// TIA Portal V20 export
FUNCTION_BLOCK "FB_LaserMeasureZoneSwitch"   // FB417, SCL
{ S7_Optimized_Access := 'TRUE' }
// stored: AutoNumber false, MemoryReserve 100, SetENOAutomatically false
   VAR RETAIN
      sMeasure1 : Bool;   // Limit sw Measure 1 / Axes are on Area Measure station 1
      sMeasure2 : Bool;   // Limit sw Measure 2 / Axes are on Area Measure station 2
      sLaser1 : Bool;   // Condition Laser 1 / Gate for going to area laser Station 1
      sLaser2 : Bool;   // Condition Laser 2 / Gate for going to area laser Station 2
      sLaserArea1Req : Bool;   // Laser area 1 request / Ask for going to laser Area Station 1
      sLaserArea2Req : Bool;   // Laser area 2 request / Ask for going to laser Area Station 2
      sCuttingArea1Req : Bool;   // Cutting 1 request / Axe X1 enter to laser Area
      sCuttingArea2Req : Bool;   // Cutting 2 request / Axe X2 enter to laser Area
      sCutBusy : Bool;   // ???
      sCut1 : Bool;   // Axe X1 traverse the gate (X1SoftLimMin1)
      sCut2 : Bool;   // Axe X2 traverse the gate (X1SoftLimMin1)
      sX1Pos : Real;
      sX2Pos : Real;
   END_VAR
   VAR
      sRT_GateCut1 : R_TRIG;
      sRT_GateCut2 : R_TRIG;
   END_VAR
   VAR RETAIN
      sCondDegageAxe : Bool;
      sRefAxisActive : Bool;
   END_VAR
BEGIN
   REGION Description header 
       //==================================================================================
       // POSALUX Swiss SA / (C) Copyright 2025
       //----------------------------------------------------------------------------------
       // Title: FB_ManageLaserOrMeasureArea
       // Comment/Function: manages two zones (laser or measurement) on two statio
       // ns, if
       // present, based on the position of the axes and/or the state of a keyboard button.
       //It dynamically switches the software limits OF the axes (limit 1 OR 2) according
       //TO the active zone, allowing the machine’s safety AND behavior TO adapt TO each
       //operating mode.
       // Author: Fabien Waldt
       // Engineering: TIA Portal v17
       //----------------------------------------------------------------------------------
       // Change log table:
       // Version  | Date     | Expert in charge | Changes applied
       // ---------|----------|------------------|------------------------------------
       // 00.00.01 | 20250224 | FWA              | First released version
       // ==================================================================================
   END_REGION

   REGION Key [16] Disable + Toggle
       // Disable Key [16] - collision detection of the ZL axis with the X axis // WFA ??
       "DB_McpKeyboardSignals".sAx10_LaserArea.sKeyDisable := NOT "LBP_ModeGroup".E_JOG;
       //On channel change, update the MCP button to reflect the toggle status of the newly selected channel 
       // "DB_McpKeyboardSignals".Ax10_LaserArea.KeySWToggleStatus :=
       // (#LaserArea1Req AND "DB_DecodChannels".Chan1IsDisplayed);
   END_REGION

   REGION Laser Area 1 Request
       IF "LBP_Chan1".MDyn[60]     // M60: Axes Limit for Laser Area
           OR ("DB_McpKeyboardSignals".sAx10_LaserArea.sKeySWTogglePositiveFront  AND "DB_DecodChannels".sChan1IsDisplayed) THEN
           #sLaserArea1Req := TRUE;
           "LBP_AlarmMsgs".ChanA[1].RID_5C02xx[0] := TRUE;         // Msg: "510200 - Waiting gate laser - M60"
       END_IF;

       IF "LBP_Chan1".MDyn[61]     // M61: Axes Limit for Measure Area
           OR ("DB_McpKeyboardSignals".sAx10_LaserArea.sKeySWToggleNegativeFront AND "DB_DecodChannels".sChan1IsDisplayed) THEN
           #sLaserArea1Req := FALSE;
           "LBP_AlarmMsgs".ChanA[1].RID_5C02xx[1] := TRUE;    // Msg: "510201 - Waiting gate measure - M61"
       END_IF;


   END_REGION

   REGION Conditions to switch the limit of axis
       IF #sLaserArea1Req 
           AND ("DB_AxisPosition".sAxis03_ZM."$AA_IM" >= "DB_AxisPosition".sAxis03_ZM."$MA_POS_LIMIT_MINUS2")  // ZM upper as limit M2
           AND ("DB_AxisPosition".sAxis04_B."$AA_IM" >= "DB_AxisPosition".sAxis04_B."$MA_POS_LIMIT_MINUS2")    // B upper as limit M2
           AND ("DB_AxisPosition".sAxis07_V."$AA_IM" <= "DB_AxisPosition".sAxis07_V."$MA_POS_LIMIT_PLUS2")     // V below as limit P2
           AND ("DB_AxisPosition".sAxis02_Y."$AA_IM" <= "DB_AxisPosition".sAxis02_Y."$MA_POS_LIMIT_PLUS2")     // Y below as limit P2
           AND "DB_Powermeter".sPowermeterInHomePos THEN   // Powermeter retracted
               #sLaser1 := TRUE;    // Set Laser 1
               #sMeasure1 := FALSE;
      ELSIF NOT #sLaserArea1Req AND
          ("DB_AxisPosition".sAxis01_X."$AA_IM" <= "DB_AxisPosition".sAxis01_X."$MA_POS_LIMIT_PLUS") THEN   // X below as limit P1
               #sMeasure1 := TRUE;
               #sLaser1 := FALSE;
       ELSE
           #sMeasure1 := FALSE;
       END_IF;
   END_REGION

   REGION Switch of the limit of axis (laser --> limit 2 / Measure --> Limit 1)
       IF #sLaser1 THEN
           "LBP_Axis01_X".A_SWLimit2Plus := TRUE;
           "LBP_Axis02_Y".A_SWLimit2Plus := TRUE;
           "LBP_Axis03_ZM".A_SWLimit2Plus := TRUE;
           "LBP_Axis04_B".A_SWLimit2Plus := TRUE;
           "LBP_Axis07_V".A_SWLimit2Plus := TRUE;
       ELSIF #sMeasure1 THEN
           "LBP_Axis01_X".A_SWLimit2Plus := FALSE;
           "LBP_Axis02_Y".A_SWLimit2Plus := FALSE;
           "LBP_Axis03_ZM".A_SWLimit2Plus := FALSE;
           "LBP_Axis04_B".A_SWLimit2Plus := FALSE;
           "LBP_Axis07_V".A_SWLimit2Plus := FALSE;
       END_IF;
   END_REGION

   REGION Led of the MCP button

       "DB_McpKeyboardSignals".sAx10_LaserArea.sLedSWStatus :=
       ((#sLaserArea1Req AND #sLaser1)
       OR (#sLaserArea1Req AND NOT #sLaser1 AND "Clock_1Hz")
       OR (NOT #sLaserArea1Req AND NOT #sLaser1 AND "Clock_1Hz"))
       AND "DB_DecodChannels".sChan1IsDisplayed
       OR ((#sLaserArea2Req AND #sLaser2)
       OR (#sLaserArea2Req AND NOT #sLaser2 AND "Clock_1Hz")
       OR (NOT #sLaserArea2Req AND NOT #sLaser2 AND "Clock_1Hz"))
       AND "DB_DecodChannels".sChan2IsDisplayed;
   END_REGION

   REGION Read in disable
       // Read in disable: laser 1 : gate NOT ready
       IF NOT #sLaserArea1Req OR #sLaser1 OR "LBP_Chan1".A_Reset THEN
           "LBP_AlarmMsgs".ChanA[1].RID_5C02xx[0] := FALSE;
       END_IF;
       IF #sLaserArea1Req OR #sMeasure1 OR "LBP_Chan1".A_Reset THEN
           "LBP_AlarmMsgs".ChanA[1].RID_5C02xx[1] := FALSE;
       END_IF;
   END_REGION

   REGION Anticollision - A REVOIR LORS MISE EN ROUTE
       REGION Conditions de dégagement
           #sCondDegageAxe := "LBP_ModeGroup".E_JOG AND NOT "LBP_ModeGroup".E_REF;
       END_REGION

       REGION Machine en Ref Active
           #sRefAxisActive := "LBP_Chan1".A_Ref OR "LBP_Chan2".A_Ref;
       END_REGION

       REGION Anticollision entre X1/V1
           IF "LBP_Axis01_X".A_SWLimit2Minus// Ne sert plus a rien car 0<v<200 
               AND ("DB_AxisPosition".sAxis07_V."$AA_IM" >= 9999.9999) THEN
               "LBP_AlarmMsgs".Axis[01].FdStop[10] := TRUE;
               "LBP_AlarmMsgs".Axis[07].FdStop[10] := TRUE;
            //   "LBP_AlarmMsgs".UserA[2].A70UUxx[10] := TRUE;   // Msg: "702010 - ???"
           END_IF;
           //Pas compris pour eviter collision avec x1 et v1
           IF (#sCondDegageAxe AND "LBP_Axis07_V".E_TCMinus)
               OR NOT "DB_DataToSafety".FrontDoorLock
               OR #sRefAxisActive THEN
               "LBP_AlarmMsgs".Axis[01].FdStop[10] := FALSE;
               "LBP_AlarmMsgs".Axis[07].FdStop[10] := FALSE;
            //   "LBP_AlarmMsgs".UserA[2].A70UUxx[10] := FALSE;   // Msg: "702010 - ???"
           END_IF;
       END_REGION

       REGION Anticollision entre X1/ZM1
           IF "LBP_Axis01_X".A_SWLimit2Minus // Ne sert plus a rien car -22<ZM1<160 
               AND (9999.9999 <= "DB_AxisPosition".sAxis03_ZM."$AA_IM") THEN
               "LBP_AlarmMsgs".Axis[01].FdStop[10] := TRUE;
               "LBP_AlarmMsgs".Axis[03].FdStop[10] := TRUE;
            //   "LBP_AlarmMsgs".UserA[2].A70UUxx[11] := TRUE;   // Msg: "702011 - ???"
           END_IF;
           //Pas compris pour eviter collision avec x1 et v1
           IF (#sCondDegageAxe AND "LBP_Axis03_ZM".E_TCPlus)
               OR NOT "DB_DataToSafety".FrontDoorLock
               OR #sRefAxisActive THEN
               "LBP_AlarmMsgs".Axis[01].FdStop[10] := FALSE;
               "LBP_AlarmMsgs".Axis[03].FdStop[10] := FALSE;
          //   "LBP_AlarmMsgs".UserA[2].A70UUxx[11] := FALSE;   // Msg: "702011 - ???"
           END_IF;
       END_REGION
   END_REGION

   REGION Cutting
       // WFA VOIR SI CUTTING NECESSAIRE POUR MACHINE MONO
       REGION Cutting : M62 waiting laser cutting free
           IF "LBP_Chan1".MDyn[62] THEN    // M62: Axes Limit for Cutting Area
               #sCuttingArea1Req := TRUE;
               "LBP_AlarmMsgs".ChanA[1].RID_5C02xx[2] := TRUE;         // Msg: "510202 - Waiting laser"
               #sX1Pos := LREAL_TO_REAL("DB_AxisPosition".sAxis01_X."$AA_IM");
           END_IF;
       END_REGION

       REGION Set cutting busy by X pos : JOG, man, prog interrupt, prog err
           #sRT_GateCut1(CLK := "DB_AxisPosition".sAxis01_X."$AA_IM" < "DB_AxisPosition".sAxis01_X."$A1_M_FP_POS4_30600");
           IF #sRT_GateCut1.Q THEN
               #sCut1 := TRUE;
           END_IF;
       END_REGION

       REGION X collision avoid
           IF #sCut1 AND #sCut2 THEN
               "LBP_AlarmMsgs".Axis[1].FdStop[0] := TRUE;
               "LBP_AlarmMsgs".Axis[10].FdStop[0] := TRUE;
           END_IF;

           // X1 plus: R stop X1
           IF "LBP_Chan1".E_ChanReset
               OR "LBP_Axis01_X".E_TCPlus
               OR "LBP_Chan1".A_Reset
               OR ("LBP_ModeGroup".E_JOG AND "LBP_ModeGroup".E_REF) THEN
               "LBP_AlarmMsgs".Axis[1].FdStop[0] := FALSE;
           END_IF;
           //check programmed X destination position
           //if in cuting area without gate_cut:stop
       END_REGION

       REGION Open cutting laser gate
           IF #sCuttingArea1Req THEN
               #sCut1 := TRUE;
               // ZL Get -> chan 1
               "LBP_Axis09_ZL".A_NCASpStrobe := TRUE;
               "LBP_Axis09_ZL".A_NCASpChanB := FALSE;
               "LBP_Axis09_ZL".A_NCASpChanA := TRUE;
           END_IF;
       END_REGION
       REGION Reset Gate_Cut_1 and Gate_Cut_2
           IF #sX1Pos >= "DB_AxisPosition".sAxis01_X."$A1_M_FP_POS4_30600" THEN
               #sX1Pos := LREAL_TO_REAL("DB_AxisPosition".sAxis01_X."$A1_M_FP_POS4_30600");
           END_IF;

           IF #sX1Pos + 1.0 < "DB_AxisPosition".sAxis01_X."$AA_IM" OR
               "LBP_Chan1".MDyn[63] THEN
               #sCut1 := FALSE;
           END_IF;
       END_REGION

       REGION Release M62
           // IF #sCut1 AND
           //     "LBP_Axis09_ZL".E_NCASpChanA
           //     AND NOT "LBP_Axis09_ZL".E_NCASpChanB
           //     OR "LBP_Chan1".A_Reset THEN
           //     "LBP_Axis09_ZL".A_NCASpStrobe := FALSE;
           //     #sCuttingArea1Req := FALSE;
           IF "DB_OPC_Laser".Scanner.In.Ready THEN
               "LBP_AlarmMsgs".ChanA[1].RID_5C02xx[2] := FALSE;         // Msg: "510202 - Waiting laser"
           END_IF;
       END_REGION
   END_REGION
   //Copie de la FL0125, Pas sur que ca existe sur les FEMTO 5A mono ou twin
   //A voir egalement les colisions à partir du code de la FL0107

   // REGION NETWORK 34
   //     IF "LBP_Chan1".MDyn[62] THEN    // M62: Axes Limit for Cutting Area
   //         #CuttingArea1Req := TRUE;
   //         "LBP_AlarmMsgs".ChanA[1].RID_5C02xx[2] := TRUE;
   //         #X1_POS := LREAL_TO_REAL("DB_AxisPosition_ReadVar".sAxis01_X1."$AA_IM");
   //     END_IF;

   //     IF "LBP_Chan2".MDyn[62] THEN    // M62: Axes Limit for Cutting Area
   //         #CuttingArea2Req := TRUE;
   //         "LBP_AlarmMsgs".ChanA[2].RID_5C02xx[2] := TRUE;
   //         #X2_POS := LREAL_TO_REAL("DB_AxisPosition_ReadVar".sAxis10_X2."$AA_IM");
   //     END_IF;
   // END_REGION

   // REGION NETWORK 35
   //     // WFA A REVOIR
   //     #Gate_Cut_1 := FALSE;
   //     #Gate_Cut_2 := FALSE;
   // END_REGION

   // REGION NETWORK 36
   //     IF #Gate_Cut_1 AND #Gate_Cut_2 THEN
   //         "LBP_AlarmMsgs".Axis[1].FdStop[0] := TRUE;
   //         "LBP_AlarmMsgs".Axis[10].FdStop[0] := TRUE;
   //     END_IF;

   //     //x1 plus: R stop x1
   //     IF "LBP_Chan1".E_ChanReset
   //         OR "LBP_Axis01_X1".E_TCPlus
   //         OR "LBP_Chan1".A_Reset
   //         OR ("LBP_ModeGroup".E_JOG AND "LBP_ModeGroup".E_REF) THEN
   //         "LBP_AlarmMsgs".Axis[1].FdStop[0] := FALSE;
   //     END_IF;

   //     //x2 minus: R stop x2
   //     IF "LBP_Chan2".E_ChanReset
   //         OR "LBP_Axis10_X2".E_TCMinus
   //         OR "LBP_Chan2".A_Reset
   //         OR ("LBP_ModeGroup".E_JOG AND "LBP_ModeGroup".E_REF) THEN
   //         "LBP_AlarmMsgs".Axis[10].FdStop[0] := FALSE;
   //     END_IF;


   //     //check programmed X destination position
   //     //if in cuting area without gate_cut:stop
   // END_REGION

   // REGION NETWORK 37
   //     IF #CuttingArea1Req AND NOT #Gate_Cut_2 THEN
   //         #Gate_Cut_1 := TRUE;
   //         "LBP_Axis09_ZL".A_NCASpStrobe := TRUE;
   //         "LBP_Axis09_ZL".A_NCASpChanB := FALSE;
   //         "LBP_Axis09_ZL".A_NCASpChanA := TRUE;
   //     END_IF;

   //     IF #CuttingArea2Req AND NOT #Gate_Cut_2 THEN
   //         #Gate_Cut_2 := TRUE;
   //         "LBP_Axis09_ZL".A_NCASpStrobe := TRUE;
   //         "LBP_Axis09_ZL".A_NCASpChanB := TRUE;
   //         "LBP_Axis09_ZL".A_NCASpChanA := FALSE;
   //     END_IF;
   // END_REGION

   // REGION NETWORK 38
   //     // WFA A REVOIR
   //     IF #X1_POS + 1.0 < "DB_AxisPosition_ReadVar".sAxis01_X1."$AA_IM" OR
   //         "LBP_Chan1".MDyn[63] THEN
   //         #Gate_Cut_1 := FALSE;
   //     END_IF;

   //     IF #X2_POS + 1.0 < "DB_AxisPosition_ReadVar".sAxis10_X2."$AA_IM" OR
   //         "LBP_Chan2".MDyn[63] THEN
   //         #Gate_Cut_2 := FALSE;
   //     END_IF;
   // END_REGION


   // REGION NETWORK 39
   //     IF #Gate_Cut_1 AND
   //         "LBP_Axis09_ZL".E_NCASpChanA
   //         AND NOT "LBP_Axis09_ZL".E_NCASpChanB
   //         OR "LBP_Chan1".A_Reset THEN
   //         "LBP_Axis09_ZL".A_NCASpStrobe := FALSE;
   //         #CuttingArea1Req := FALSE;
   //         "LBP_AlarmMsgs".ChanA[1].RID_5C02xx[2] := FALSE;
   //     END_IF;

   //     IF #Gate_Cut_2 AND
   //         NOT "LBP_Axis09_ZL".E_NCASpChanA
   //         AND "LBP_Axis09_ZL".E_NCASpChanB
   //         OR "LBP_Chan2".A_Reset THEN
   //         "LBP_Axis09_ZL".A_NCASpStrobe := FALSE;
   //         #CuttingArea2Req := FALSE;
   //         "LBP_AlarmMsgs".ChanA[2].RID_5C02xx[2] := FALSE;
   //     END_IF;
   // END_REGION
END_FUNCTION_BLOCK
